// TIA Portal project "PLC1500与无刷驱动控制" (V14)

(* hardware
DEVICE "S71500/ET200MP station_1"  S7-1500 station
   slot 0: "导轨_0"  Rack  6ES7 590-1***0-0AA0
   slot 1: "PLC_1"  CPU 1516-3 PN/DP  6ES7 516-3AN01-0AB0  V2.1
      slot 3: "CPU 显示_1"  6ES7591-1BA00-0AA0
   slot 2: "DI 32x24VDC HF_1"  DI 32x24VDC HF  6ES7 521-1BL00-0AB0  V2.1
   slot 3: "DQ 32x24VDC/0.5A HF_1"  DQ 32x24VDC/0.5A HF  6ES7 522-1BL01-0AB0  V1.0
   slot 4: "AI 8xU/I/RTD/TC ST_1"  AI 8xU/I/RTD/TC ST  6ES7 531-7KF00-0AB0  V2.1
   slot 5: "AQ 4xU/I ST_1"  AQ 4xU/I ST  6ES7 532-5HD00-0AB0  V2.1
*)

// ===== PLC "PLC_1"  CPU 1516-3 PN/DP =====

VAR_GLOBAL   // PLC tag table "无刷电机IO"
   "无刷电机正转" AT %Q1.1 : Bool;
   "无刷电机反转" AT %Q1.2 : Bool;
   "无刷电机速度M0" AT %Q1.3 : Bool;
   "无刷电机速度M1" AT %Q1.4 : Bool;
   "无刷电机速度设定" AT %QW4 : Word;
END_VAR

DATA_BLOCK "无刷电机驱动控制"   // DB1
{ S7_Optimized_Access := 'TRUE' }
VERSION : 0.1
   VAR
      正转启动 : Bool;
      反转启动 : Bool;
      速度M0 : Bool;
      速度M1 : Bool;
      速度设定 : Int;
      Speed_Temp : Real;
   END_VAR
BEGIN
END_DATA_BLOCK

ORGANIZATION_BLOCK "Main"   // OB1, LAD, ProgramCycle
TITLE = "Main Program Sweep (Cycle)"
{ S7_Optimized_Access := 'TRUE' }
VERSION : 0.1
   VAR_INPUT
      Initial_Call : Bool;   // Initial call of this OB
      Remanence : Bool;   // =True, if remanent data are available
   END_VAR
BEGIN

REGION Network 1: 正转启动
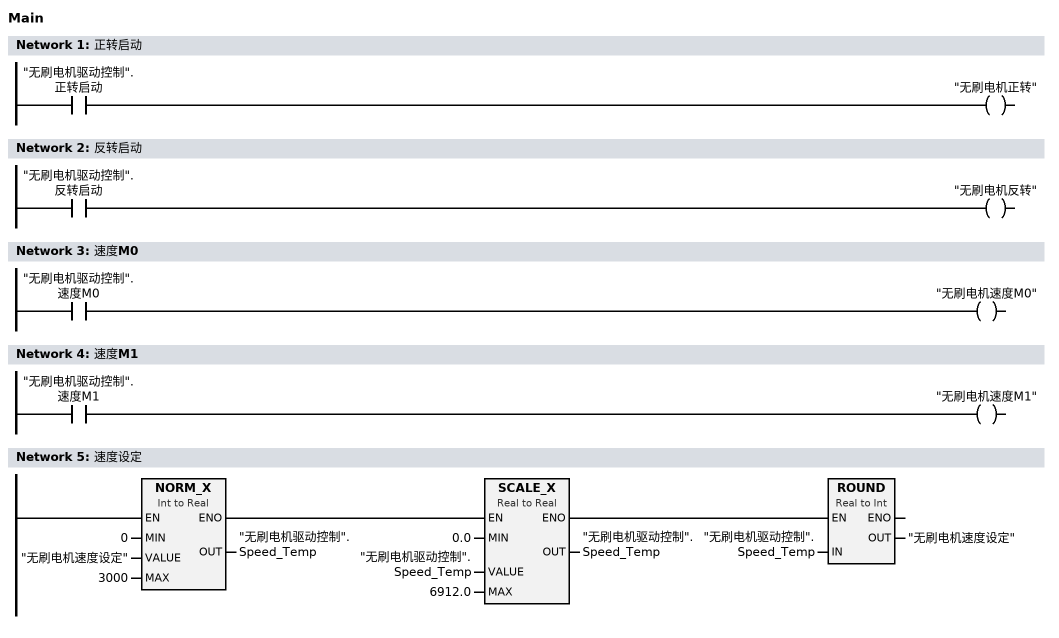
   RUNG wire#powerrail
      Contact( "无刷电机驱动控制".正转启动 )
      Coil( "无刷电机正转" )
   END_RUNG
   // the same network as SCL:
   "无刷电机正转" := "无刷电机驱动控制".正转启动;
END_REGION

REGION Network 2: 反转启动
   RUNG wire#powerrail
      Contact( "无刷电机驱动控制".反转启动 )
      Coil( "无刷电机反转" )
   END_RUNG
   // the same network as SCL:
   "无刷电机反转" := "无刷电机驱动控制".反转启动;
END_REGION

REGION Network 3: 速度M0
   RUNG wire#powerrail
      Contact( "无刷电机驱动控制".速度M0 )
      Coil( "无刷电机速度M0" )
   END_RUNG
   // the same network as SCL:
   "无刷电机速度M0" := "无刷电机驱动控制".速度M0;
END_REGION

REGION Network 4: 速度M1
   RUNG wire#powerrail
      Contact( "无刷电机驱动控制".速度M1 )
      Coil( "无刷电机速度M1" )
   END_RUNG
   // the same network as SCL:
   "无刷电机速度M1" := "无刷电机驱动控制".速度M1;
END_REGION

REGION Network 5: 速度设定
   RUNG wire#powerrail
      { S7_Templates := "[SrcType := Int, DestType := Real]" } Normalize(min := 0, value := "无刷电机速度设定", max := 3000, out => "无刷电机驱动控制".Speed_Temp)
      { S7_Templates := "[SrcType := Real, DestType := Real]" } Scale(min := 0.0, value := "无刷电机驱动控制".Speed_Temp, max := 6912.0, out => "无刷电机驱动控制".Speed_Temp)
      { S7_Templates := "[SrcType := Real, DestType := Int]" } Round(in := "无刷电机驱动控制".Speed_Temp, out => "无刷电机速度设定")
   END_RUNG
   // the same network as SCL:
   "无刷电机驱动控制".Speed_Temp := NORM_X(MIN := 0, VALUE := "无刷电机速度设定", MAX := 3000);
   "无刷电机驱动控制".Speed_Temp := SCALE_X(MIN := 0.0, VALUE := "无刷电机驱动控制".Speed_Temp, MAX := 6912.0);
   "无刷电机速度设定" := ROUND("无刷电机驱动控制".Speed_Temp);
END_REGION
END_ORGANIZATION_BLOCK